FUNCTION_BLOCK CU040ManualTask EXTENDS TcoTaskedService IMPLEMENTS ICUTask
VAR
END_VAR

Run();

(*~
	<docu>
		<summary>
			Main method of the sequener. Custom code needs to be placed here. The sequencer is executed by call of **Instance.Run()** method.
			This method is abstract, and it must be overridden in derived block.
		</summary>
	</docu>
~*)
METHOD PROTECTED Main : BOOL
Messenger.Notify('Running manual mode');
Station.Components.Group1.horizontalCylinder.Service();
END_METHOD

METHOD PROTECTED OnStart
Station.AutomatTask.Restore();
Station.GroundTask.Restore();
Station.GroundTask.CancelGround();
END_METHOD

PROPERTY Station : REFERENCE TO CU040
GET
VAR
    _station : POINTER TO CU040;
END_VAR
IF __QUERYPOINTER(Parent, _station) THEN // Check if _Parent is Station001
    Station REF= _station^;              // If the check is successful dereference a pointer. simlar to THIS^ or SUPER^
END_IF
END_GET
END_PROPERTY

END_FUNCTION_BLOCK

(* stored: Version 1.1.0.1
   POU CU040ManualTask: Id {2203494c-e440-43e1-b2da-8abbda7d7511}, SpecialFunc None
   Method Main: Id {6c71b746-70b9-4223-90f3-a350683250a5}
   Method OnStart: Id {2b52ea36-1277-4f28-968d-9c0eaaba55fd}
   Property Station: Id {068d8939-9783-4a05-8f45-03edef15128b}
   Get Get: Id {7e39b1e6-c366-4977-9f30-424ac7d23757} *)
